FUNCTION_BLOCK FB_DateAndTimeHandling
VAR_INPUT
END_VAR
VAR_OUTPUT
END_VAR
VAR
	
	
	TimeStruct :					Tc2_Utilities.TIMESTRUCT;
	fbGetTime:						NT_GetTime;
	
	GetTimeTON :					TON;	

END_VAR

METHOD Enable : BOOL
VAR_INPUT
END_VAR
fbGetTime(
	NETID:='' , 
	START:= GetTimeTON.Q, 
	TMOUT:= T#40S , 
	TIMESTR=>TimeStruct );
END_METHOD

PROPERTY GetActualDayOfMonthAsINT : INT
GET
GetActualDayOfMonthAsINT := WORD_TO_INT(TimeStruct.wDay);
END_GET
END_PROPERTY

PROPERTY GetActualHourAsINT : INT
GET
GetActualHourAsINT := WORD_TO_INT(TimeStruct.wHour);
END_GET
END_PROPERTY

PROPERTY GetActualMillisecondAsINT : INT
GET
GetActualMillisecondAsINT := WORD_TO_INT(TimeStruct.wMilliseconds);
END_GET
END_PROPERTY

PROPERTY GetActualMinuteAsINT : INT
GET
GetActualMinuteAsINT := WORD_TO_INT(TimeStruct.wMinute);
END_GET
END_PROPERTY

PROPERTY GetActualMonthAsINT : INT
GET
GetActualMonthAsINT := WORD_TO_INT(TimeStruct.wMonth);
END_GET
END_PROPERTY

PROPERTY GetActualSecondAsINT : INT
GET
GetActualSecondAsINT := WORD_TO_INT(TimeStruct.wSecond);
END_GET
END_PROPERTY

PROPERTY GetActualWeekdayAsINT : INT
GET
GetActualWeekdayAsINT := WORD_TO_INT(TimeStruct.wDayOfWeek);
END_GET
END_PROPERTY

PROPERTY GetActualYearAsINT : INT
GET
GetActualYearAsINT := WORD_TO_INT(TimeStruct.wYear);
END_GET
END_PROPERTY

PROPERTY GetDateAsSTRING : STRING
GET
VAR
	
	DateTime :						DT;
	ToUDT :							STRING;
	WithOutDT :						STRING;
	WithOutHyphen :					STRING;
	WithGap :						STRING;
	DateTimeString :				STRING;
	TimeString :					STRING;	

END_VAR
//Date To String
	//Makes TimeStruct to DateTime
	DateTime := SYSTEMTIME_TO_DT(TIMESTR:= TimeStruct);
	
	//Makes DateTime to String
	ToUDT := DT_TO_STRING(DateTime);
	
	//Delete #DT from String
	WithOutDT := Tc2_Standard.DELETE(STR:=ToUDT, LEN:=4,POS:=0);
	
	//Delete hyphen between date and time
	WithOutHyphen:=Tc2_Standard.DELETE(STR:=WithOutDT, LEN:=1,POS:=11);
	
	//Insert a gap between date and time	
	WithGap := Tc2_Standard.INSERT(STR1:=WithOutHyphen,STR2:=' ', POS:=10);
	DateTimeString := Tc2_Standard.DELETE(STR:=WithGap, LEN:=6,POS:=0);
	GetDateAsSTRING := Tc2_Standard.DELETE(STR:=DateTimeString, LEN:=7,POS:=8);
END_GET
END_PROPERTY

PROPERTY GetDateTimeAsSTRING : STRING
GET
VAR

	DateTime :						DT;
	ToUDT :							STRING;
	WithOutDT :						STRING;
	WithOutHyphen :					STRING;
	WithGap :						STRING;
	DateTimeString :				STRING;
	TimeString :					STRING;	

END_VAR
//Date To String
	//Makes TimeStruct to DateTime
	DateTime := SYSTEMTIME_TO_DT(TIMESTR:= TimeStruct);
	
	//Makes DateTime to String
	ToUDT := DT_TO_STRING(DateTime);
	
	//Delete #DT from String
	WithOutDT := Tc2_Standard.DELETE(STR:=ToUDT, LEN:=4,POS:=0);
	
	//Delete hyphen between date and time
	WithOutHyphen:=Tc2_Standard.DELETE(STR:=WithOutDT, LEN:=1,POS:=11);
	
	//Insert a gap between date and time	
	WithGap := Tc2_Standard.INSERT(STR1:=WithOutHyphen,STR2:=' ', POS:=10);
	DateTimeString := Tc2_Standard.DELETE(STR:=WithGap, LEN:=6,POS:=0);
	TimeString := Tc2_Standard.DELETE(STR:=DateTimeString, LEN:=7,POS:=0);
	GetDateTimeAsSTRING := DateTimeString;
END_GET
END_PROPERTY

PROPERTY GetRawDateTimeAsSTRING : STRING
GET
VAR
	
	DateTime :						DT;
	ToUDT :							STRING;
	WithOutDT :						STRING;
	EmptyString :					STRING(1);
	DateTimeString :				STRING;
	TimeString :					STRING;	

END_VAR
//Makes TimeStruct to DateTime
	DateTime := SYSTEMTIME_TO_DT(TIMESTR:= TimeStruct);
	
	//Makes DateTime to String
	ToUDT := DT_TO_STRING(DateTime);

	
	//Delete #DT from String
	WithOutDT := Tc2_Standard.DELETE(STR:=ToUDT, LEN:=4,POS:=0);

	//Delete hyphen between date and time
	GetRawDateTimeAsSTRING:= Tc2_Standard.REPLACE(STR1:=WithOutDT , STR2:=' ' , L:=1 , P:=11 ); //Tc2_Standard.DELETE(STR:=WithOutDT, LEN:=1,POS:=11);
END_GET
END_PROPERTY

PROPERTY GetTimeAsSTRING : STRING
GET
VAR

	DateTime :						DT;
	ToUDT :							STRING;
	WithOutDT :						STRING;
	WithOutHyphen :					STRING;
	WithGap :						STRING;
	DateTimeString :				STRING;
	TimeString :					STRING;	

END_VAR
//Date To String
	//Makes TimeStruct to DateTime
	DateTime := SYSTEMTIME_TO_DT(TIMESTR:= TimeStruct);
	
	//Makes DateTime to String
	ToUDT := DT_TO_STRING(DateTime);
	
	//Delete #DT from String
	WithOutDT := Tc2_Standard.DELETE(STR:=ToUDT, LEN:=4,POS:=0);
	
	//Delete hyphen between date and time
	WithOutHyphen:=Tc2_Standard.DELETE(STR:=WithOutDT, LEN:=1,POS:=11);
	
	//Insert a gap between date and time	
	WithGap := Tc2_Standard.INSERT(STR1:=WithOutHyphen,STR2:=' ', POS:=10);
	DateTimeString := Tc2_Standard.DELETE(STR:=WithGap, LEN:=6,POS:=0);
	GetTimeAsSTRING := Tc2_Standard.DELETE(STR:=DateTimeString, LEN:=7,POS:=0);
END_GET
END_PROPERTY

END_FUNCTION_BLOCK

(* stored: Version 1.1.0.1, ProductVersion 3.1.4024.15
   POU FB_DateAndTimeHandling: Id {db6a0d7c-3577-4ce2-a433-d0be31df9fdb}, SpecialFunc None
   Method Enable: Id {84bb056b-d454-480f-b497-6949f4858af8}
   Property GetActualDayOfMonthAsINT: Id {b5e5be76-9282-4204-9d79-3740f13f0542}
   Get Get: Id {3f9fced7-5b54-42c5-b9a8-c83a0c3dc83b}
   Property GetActualHourAsINT: Id {0af0a903-f925-47e9-bd28-84bad65f617b}
   Get Get: Id {199c8e4b-941e-44b3-9b42-76f6d8ba5a02}
   Property GetActualMillisecondAsINT: Id {316bea74-ce1b-4be4-adf5-986f22615a4e}
   Get Get: Id {12543d29-4189-4ade-9011-c2a31cf8c5cc}
   Property GetActualMinuteAsINT: Id {8b9811d3-19fc-4217-8b01-d98bd8d9ffd7}
   Get Get: Id {253aa4c1-2909-4e5a-873a-24ca345d5821}
   Property GetActualMonthAsINT: Id {ce63e3d7-c964-4307-a839-bb12b2fdf788}
   Get Get: Id {16386204-753e-4f81-997b-4c581229ef8d}
   Property GetActualSecondAsINT: Id {31c925ed-682c-450a-93de-5d070aa99fa7}
   Get Get: Id {eb3e216b-76cd-4b63-ab4a-94acd22a945c}
   Property GetActualWeekdayAsINT: Id {7022b24d-b771-499f-9e9b-9d468aada62b}
   Get Get: Id {f66592c2-a168-40de-ab9e-defa0aea60b5}
   Property GetActualYearAsINT: Id {5981dab8-27e8-4a11-b6e8-7aecaf6f3d10}
   Get Get: Id {39569eab-afab-49a9-b487-6ed23f36b4f8}
   Property GetDateAsSTRING: Id {bdd45043-adde-4bed-89fd-1aeeb7d85e26}
   Get Get: Id {f6087201-9493-4012-83db-ee84f7cdd20c}
   Property GetDateTimeAsSTRING: Id {8e9b2525-6494-4daa-acff-d34b656004b3}
   Get Get: Id {eea35a9c-5bac-466b-8075-eac3ef0d9d13}
   Property GetRawDateTimeAsSTRING: Id {c36e9886-5256-40e4-919f-8b674b133ee3}
   Get Get: Id {1dd97c43-0b5f-4a2f-ac34-74195f9ee609}
   Property GetTimeAsSTRING: Id {16d69dcc-e62e-490d-96d0-52b7d55bd6cc}
   Get Get: Id {326bb161-5757-4721-a146-3ee454039e1e} *)
